INTERFACE I_Emit

METHOD Emit
VAR_INPUT
	iArg			: Calls.I_Arg;
END_VAR
END_METHOD

METHOD EmitTo : Results.Result
VAR_INPUT
	iReceiver		: I_Receiver;
	iArg			: Calls.I_Arg;
END_VAR
END_METHOD

METHOD Option : REFERENCE TO Signal
VAR_INPUT
	sOption		: Strings.Str;
END_VAR
END_METHOD

METHOD Pair : Results.Result
VAR_INPUT
	iReceiver		: I_Receiver;
END_VAR
END_METHOD

PROPERTY Tag : Tags.I_Tag
GET
END_GET
END_PROPERTY

METHOD Unpair : Results.Result
VAR_INPUT
	iReceiver		: I_Receiver;
END_VAR
END_METHOD

END_INTERFACE

(* stored: Version 1.1.0.1
   Itf I_Emit: Id {b1e715f2-0d63-401e-ad83-c78f9a27c3e1}
   Method Emit: Id {f041e330-cb67-4705-990a-25a4d7e716bd}
   Method EmitTo: Id {f63f9e41-331e-4141-ade2-766fd1e035f1}
   Method Option: Id {2f6744b0-bd8d-42ca-819f-aa5355c15691}
   Method Pair: Id {61a365c3-bccb-4448-8e02-7787a026cdda}
   Property Tag: Id {db4a3b23-2e65-46f0-8ce7-4733479fdf10}
   Get Get: Id {81070cf0-fcb9-4d4f-80c8-9a287f1ece44}
   Method Unpair: Id {e00c6d52-6ad6-4fc6-a0ec-4c25e00bf6c6} *)
